RoboDK station: Double suction HAMK Robotics station MG400 Wood Sticks Solution Python.rdk

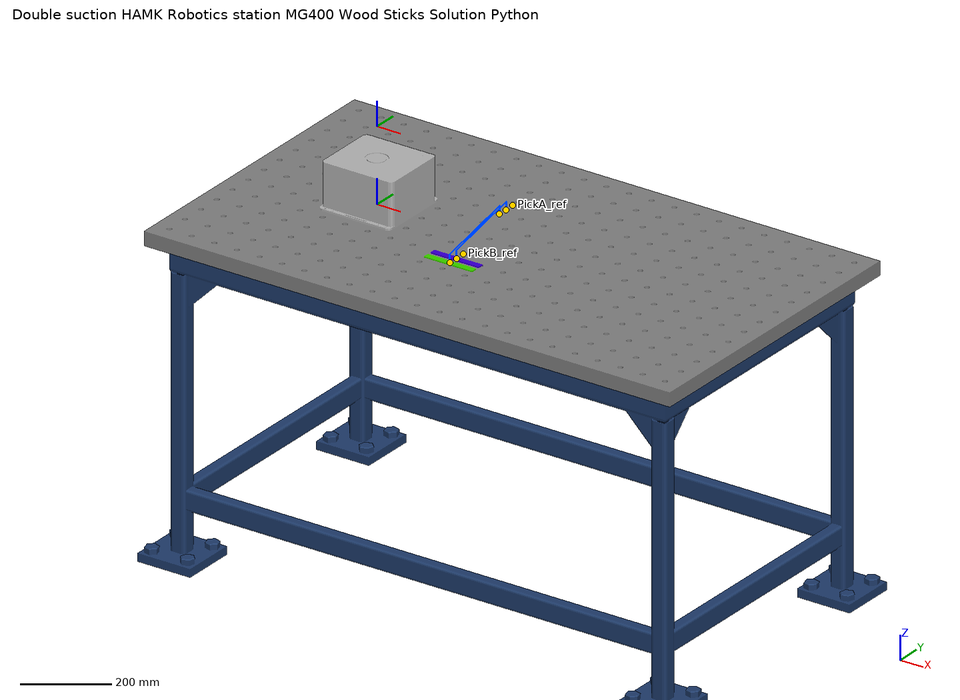
[picture v0: the station drawn from its stored meshes, robots at their saved joint values, targets as dots, program paths as lines]
Station Double suction HAMK Robotics Station MG400 Wood Sticks (saved by RoboDK 5.6.7). Poses are relative to the parent item; angles as X-Y-Z fixed-axis rotations.
Station parameters (name, value as stored): IO_1, 0, LIN64
  - frame Dobot MG400 Base at (0, 0, 0) mm
    - robot Dobot MG400: 4 axes, payload 0.5 kg, reach 393.5 mm, repeatability 0.2 mm, weight 4 kg
        joint limits [-160, -25, -25, -360] to [160, 85, 105, 360]; home [0, 0, 0, 0]; saved at [-26.564, 65.279, 67.505, -26.574]
      - tool Suction Cup, TCP at (0, 0, 75.5) mm, size 42.6 x 40 x 76.8 mm
    - frame World at (0, 0, 0) mm
      - object Table 1400x800x800mm at (0, 0, 0) mm, size 1420 x 820 x 800 mm, geometry from Table-1400x800x800mm.sld
        - object HAMK logo at (360, 380, -115) mm, rotated rx 90 ry 0 rz 180 deg, size 301.4 x 100.9 x 9.4 mm, geometry from Fantastic Duup(2).stl
        - object white background at (360, 385.5, -110) mm, rotated rx 90 ry 0 rz 0 deg, size 480 x 184.8 x 2.4 mm, geometry from Fantastic Duup(3).stl
      - object Wood Stick at (250, 160, 0) mm, rotated rx 180 ry 0 rz 180 deg, size 128 x 15 x 3 mm, geometry from Wood Stick Biltema.stl
      - object stick1 at (300, -125, 0) mm, rotated rx 180 ry 0 rz 180 deg, size 128 x 15 x 3 mm, geometry from Wood Stick Biltema.stl
      - object stick2 at (300, -150, 0) mm, rotated rx 180 ry 0 rz 180 deg, size 128 x 15 x 3 mm, geometry from Wood Stick Biltema.stl
  - frame RefSuctionCup at (0, 0, 189) mm
    - target PickA_ref (Cartesian target) at (250, 160, -186) mm, rotated rx 180 ry 0 rz -179.99 deg; joints [32.619, 68.287, 81.875, 32.609] of Dobot MG400
    - target PickB_ref (Cartesian target) at (300, -100, -186) mm, rotated rx 180 ry 0 rz -179.99 deg; joints [-18.435, 69.533, 75.852, -18.445] of Dobot MG400
    - target PickA1 (Cartesian target) at (250, 135, -186) mm, rotated rx 180 ry 0 rz -179.99 deg; joints [32.619, 68.287, 81.875, 32.609] of Dobot MG400
    - target PickA2 (Cartesian target) at (250.01, 110, -186) mm, rotated rx 180 ry 0 rz -179.99 deg; joints [32.619, 68.287, 81.875, 32.609] of Dobot MG400
    - target PickB1 (Cartesian target) at (300, -125, -186) mm, rotated rx 180 ry 0 rz -179.99 deg; joints [-18.435, 69.533, 75.852, -18.445] of Dobot MG400
    - target PickB2 (Cartesian target) at (300.01, -150, -186) mm, rotated rx 180 ry 0 rz -179.99 deg; joints [-18.435, 69.533, 75.852, -18.445] of Dobot MG400
  - Python program Create_duplicates (listed below)
  - Python program Generate_program (listed below)
  - program StartPositions (1 instructions, listed below)
  - program AutoMove (26 instructions, listed below)
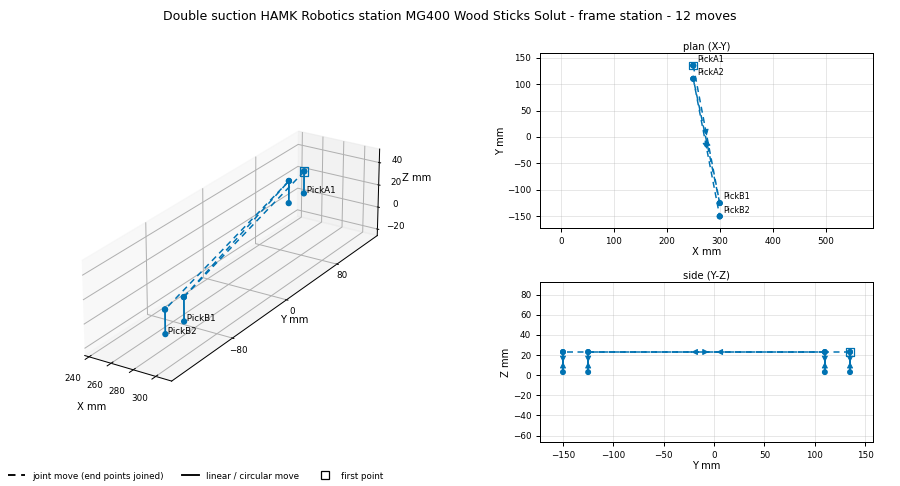
[picture p0: tool path of Double suction HAMK Robotics station MG400 Wood Sticks Solution Python.rdk in frame station, 12 of 12 moves have a stored position in this frame; points joined in program order, loops and branches not executed]

--- Python program Create_duplicates ---
# Duplicate objects
#
# Fernando Pacheco
# 2024-01

OBJWIDTH = 15
CLEARANCE = 10 # separation between objects

from robodk import robolink    # RoboDK API
from robodk import robomath    # Robot toolbox
RDK = robolink.Robolink()

# Locate the reference box
item = RDK.Item('Wood Stick', robolink.ITEM_TYPE_OBJECT)
if item.Valid():
    print('Item selected: ' + item.Name())
    print('Item position: ' + repr(item.Pose()))
else:
    raise Exception('Item not valid')

item.Copy() # like doing ctrl+C

# To paste, we need a reference frame
frame = RDK.Item('World', robolink.ITEM_TYPE_FRAME)
RDK.Render(False)
# paste in the frame the object
# that was previously copied
num_new = 2
step = 1.0/(num_new-1)
for i in range(num_new):
    newitem = frame.Paste()
    newitem.setName('stick'+str(i+1))
    newitem.setPose(item.Pose() * robomath.transl(0,-(OBJWIDTH+CLEARANCE)*(i+1)))
    newitem.setVisible(True, False) # item is visible, its reference frame no
    newitem.Recolor([0.3, step*i, 1 - step*i, 1])
item.setVisible(False, False) # make the reference object not visible
RDK.Render(True)

# Create source targets
item = RDK.Item('PickA_ref', robolink.ITEM_TYPE_TARGET)
item.Copy()
# for the Dobot post-processor, the reference frame should be only one
# it's not possible to change to another reference frame
# because the function to do it is not implemented
frame = RDK.Item('RefSuctionCup', robolink.ITEM_TYPE_FRAME)
RDK.Render(False)
# paste in the frame the object
# that was previously copied
for i in range(num_new):
    newitem = frame.Paste()
    newitem.setName('PickA'+str(i+1))
    newitem.setPose(item.Pose() * robomath.transl(0,-(OBJWIDTH+CLEARANCE)*(i+1)))
    newitem.setVisible(True, False) # item is visible, its reference frame no
RDK.Render(True)

# Create destination targets
item = RDK.Item('PickB_ref', robolink.ITEM_TYPE_TARGET)
item.Copy()
frame = RDK.Item('RefSuctionCup', robolink.ITEM_TYPE_FRAME)
RDK.Render(False)
# paste in the frame the object
# that was previously copied
for i in range(num_new):
    newitem = frame.Paste()
    newitem.setName('PickB'+str(i+1))
    newitem.setPose(item.Pose() * robomath.transl(0,-(OBJWIDTH+CLEARANCE)*(i+1)))
    newitem.setVisible(True, False) # item is visible, its reference frame no
RDK.Render(True)

--- Python program Generate_program ---
# Create program to run in the robot
#
# Fernando Pacheco
# 2024-01

num_new=2 # number of new objects that were created

from robodk import robolink    # RoboDK API
from robodk import robomath    # Robot toolbox
RDK = robolink.Robolink()

frame = RDK.Item('RefSuctionCup', robolink.ITEM_TYPE_FRAME)
if not frame.Valid():
    raise Exception('RefFrame RefSuctionCup is not valid')

# How to create attach and detach events
# From https://robodk.com/forum/Thread-Attach-an-object-in-python
INS_TYPE_EVENT = 7
EVENT_ATTACH = 0
EVENT_DETACH = 1
tool = RDK.Item('Suction Cup', robolink.ITEM_TYPE_TOOL)
if not tool.Valid():
    raise Exception('Tool Suction Cup is not valid')
frameWorld = RDK.Item('World', robolink.ITEM_TYPE_FRAME)
if not frameWorld.Valid():
    raise Exception('RefFrame World is not valid')
ins_event_attach = {'Type': INS_TYPE_EVENT, 'Behavior': EVENT_ATTACH, 'ToolPtr': str(tool.item)}
ins_event_detach = {'Type': INS_TYPE_EVENT, 'Behavior': EVENT_DETACH, 'ToolPtr': str(tool.item), 'FramePtr': str(frameWorld.item)}

# The program to move from targets A to targets B
prog = RDK.AddProgram('AutoMove')

prog.setPoseFrame(frame)
tool = RDK.Item('Suction Cup')
prog.setPoseTool(tool)

itemlist = RDK.ItemList(filter=robolink.ITEM_TYPE_TARGET)
for i in range(num_new):
    for item in itemlist:
        if item.Name()=='PickA'+str(i+1):
            print(f'Move PickA{i+1}')
            prog.MoveJ(item.Pose()*robomath.transl(0,0,-20))
            prog.MoveL(item)
            prog.setParam("Add",ins_event_attach) # ATTACH simulation only
            prog.setDO('1', 1) # turn ON vacuum
            prog.Pause(1000) # then wait
            prog.MoveL(item.Pose()*robomath.transl(0,0,-20)) # go up first
    for item in itemlist:
        if item.Name()=='PickB'+str(i+1):
            prog.MoveJ(item.Pose()*robomath.transl(0,0,-20))
            prog.MoveL(item)
            prog.setParam("Add",ins_event_detach) # DETACH simulation only
            prog.setDO('1', 0) # turn OFF vacuum
            prog.Pause(1000) # then wait
            prog.MoveL(item.Pose()*robomath.transl(0,0,-20))

--- program StartPositions (robot Dobot MG400) ---
  Replace objects

--- program AutoMove (robot Dobot MG400) ---
  Set Ref.: RefSuctionCup
  Set Tool: Suction Cup
  MoveJ 2 to (250, 135, -166) mm, rotated rx 180 ry 0 rz -179.99 deg; joints [28.369, 60.886, 82.865, 28.359]
  MoveL (PickA1)
  Attach to Suction Cup
  Set IO_1=1
  Pause 1.0 s
  MoveL 7 to (250, 135, -166) mm, rotated rx 180 ry 0 rz -179.99 deg; joints [28.369, 60.886, 82.865, 28.359]
  MoveJ 8 to (300, -125, -166) mm, rotated rx 180 ry 0 rz -179.99 deg; joints [-22.62, 64.056, 70.596, -22.63]
  MoveL (PickB1)
  Detach from Suction Cup
  Set IO_1=0
  Pause 1.0 s
  MoveL 13 to (300, -125, -166) mm, rotated rx 180 ry 0 rz -179.99 deg; joints [-22.62, 64.056, 70.596, -22.63]
  MoveJ 14 to (250.01, 110, -166) mm, rotated rx 180 ry 0 rz -179.99 deg; joints [23.749, 60.515, 86.297, 23.739]
  MoveL (PickA2)
  Attach to Suction Cup
  Set IO_1=1
  Pause 1.0 s
  MoveL 19 to (250.01, 110, -166) mm, rotated rx 180 ry 0 rz -179.99 deg; joints [23.749, 60.515, 86.297, 23.739]
  MoveJ 20 to (300.01, -150, -166) mm, rotated rx 180 ry 0 rz -179.99 deg; joints [-26.564, 65.279, 67.505, -26.574]
  MoveL (PickB2)
  Detach from Suction Cup
  Set IO_1=0
  Pause 1.0 s
  MoveL 25 to (300.01, -150, -166) mm, rotated rx 180 ry 0 rz -179.99 deg; joints [-26.564, 65.279, 67.505, -26.574]
